(* CODESYS project TeSTL_RECOVERED_2026-06-30T05-16-33.project

Project tree, tasks and I/O mapping:
  Device : CODESYS Control Win V3 x64, CODESYS, version 3.5.22.20
    application Application
      libraries: Standard, 3.5.22.0 (System)
      task MainTask (cyclic, interval t#20ms, priority 1) calls PLC_PRG
      program PLC_PRG [ST]
*)

// Device/Application/PLC_PRG
PROGRAM PLC_PRG
VAR
    // ---- PHYSICAL INPUTS (Mapped to IO Modules) ----
    xProximitySensor     : BOOL;  // Detects a part arriving at the inspection point
    xPartInBin1Sensor    : BOOL;  // Verification sensor for Bin 1
    xPartInBin2Sensor    : BOOL;  // Verification sensor for Bin 2
    xPartInRejectSensor  : BOOL;  // Verification sensor for Reject Bin
    
    // ---- PHYSICAL OUTPUTS (Mapped to Relays/Actuators) ----
    xMainConveyorMotor   : BOOL;  // High-voltage motor running the belt
    xPusherActuator1     : BOOL;  // Pneumatic piston for Bin 1
    xPusherActuator2     : BOOL;  // Pneumatic piston for Bin 2
    
    // ---- RASPBERRY PI NETWORK INTERFACE (Modbus/EtherNET IP Map) ----
    // The Pi writes to these registers
    xPi_Heartbeat        : BOOL;  // Toggle bit to monitor if the Pi is alive
    xPi_NewInstruction   : BOOL;  // Strobe bit signaling a routing decision is ready
    diPi_TargetBin       : DINT;  // Target Destination: 1 = Bin 1, 2 = Bin 2, 3 = Reject
    
    // The PLC writes to these registers for the Pi to read
    xPLC_PartReadyForScan: BOOL;  // Signals the Pi to run its Computer Vision/Camera script
    xPLC_SystemReady     : BOOL;  // System health indicator
    xPLC_ErrorFault      : BOOL;  // Active fault indicator
    
    // ---- INTERNAL CONTROL LOGIC & STATE MACHINE ----
    iSystemState         : INT := 0;   // Main State Machine Step counter
    diAssignedRoute      : DINT;       // Latched routing destination for current part
    tonPusherTimeout     : TON;        // Built-in Timer for Actuator extension
    tonWatchdog          : TON;        // Heartbeat Watchdog Timer for Raspberry Pi communication
    xLastPiHeartbeatState: BOOL;  // Memory flag to track edge transitions of the heartbeat
END_VAR

// ==========================================
// 1. SAFETY & COMMUNICATION WATCHDOG
// ==========================================
// Track if the Raspberry Pi stops communicating. 
// If xPi_Heartbeat doesn't toggle state within 3.0 seconds, trigger a fault.

tonWatchdog(IN := (xPi_Heartbeat = xLastPiHeartbeatState), PT := T#3S);

IF tonWatchdog.Q THEN
    xPLC_ErrorFault := TRUE;
    iSystemState := 99; // Jump straight to Emergency / Fault State
END_IF;

xLastPiHeartbeatState := xPi_Heartbeat; // Store current state for next cyclic scan


// ==========================================
// 2. MAIN SORTING STATE MACHINE
// ==========================================
CASE iSystemState OF
    
    0: (* STATE 0: System Initialization & Idle State *)
        xMainConveyorMotor   := FALSE;
        xPusherActuator1     := FALSE;
        xPusherActuator2     := FALSE;
        xPLC_PartReadyForScan:= FALSE;
        xPLC_SystemReady     := TRUE;
        
        IF NOT xPLC_ErrorFault THEN
            xMainConveyorMotor := TRUE; // Start conveyor if safe
            iSystemState := 10;
        END_IF;

    10: (* STATE 10: Wait for Part Arrival *)
        IF xProximitySensor THEN
            xMainConveyorMotor := FALSE;      // Halt conveyor to take clean camera frame
            xPLC_PartReadyForScan := TRUE;    // Strobe signal to Raspberry Pi
            iSystemState := 20;
        END_IF;

    20: (* STATE 20: Wait for Raspberry Pi Decision Handshake *)
        // Pi processes image -> Writes destination register -> Sets xPi_NewInstruction TRUE
        IF xPi_NewInstruction THEN
            diAssignedRoute := diPi_TargetBin; // Latch the routing decision locally
            xPLC_PartReadyForScan := FALSE;    // Lower the request flag
            xMainConveyorMotor := TRUE;        // Resume conveyor movement
            iSystemState := 30;
        END_IF;

    30: (* STATE 30: Execute Sorting Trajectory *)
        CASE diAssignedRoute OF
            1: (* Route to Bin 1 *)
                xPusherActuator1 := TRUE;
                tonPusherTimeout(IN := TRUE, PT := T#1.5S); // Allow piston to fully extend
                
                IF xPartInBin1Sensor OR tonPusherTimeout.Q THEN
                    xPusherActuator1 := FALSE;
                    tonPusherTimeout(IN := FALSE); // Reset Timer
                    iSystemState := 0;             // Cycle Complete, return to idle
                END_IF;
                
            2: (* Route to Bin 2 *)
                xPusherActuator2 := TRUE;
                tonPusherTimeout(IN := TRUE, PT := T#1.5S);
                
                IF xPartInBin2Sensor OR tonPusherTimeout.Q THEN
                    xPusherActuator2 := FALSE;
                    tonPusherTimeout(IN := FALSE);
                    iSystemState := 0;
                END_IF;
                
            3: (* Route directly to default Reject Bin *)
                IF xPartInRejectSensor THEN
                    iSystemState := 0;
                END_IF;
        ELSE
            // If the Pi passes an invalid destination code, trigger a fault routing anomaly
            xPLC_ErrorFault := TRUE;
            iSystemState := 99;
        END_CASE;

    99: (* STATE 99: Emergency Fault Handling *)
        xMainConveyorMotor   := FALSE;
        xPusherActuator1     := FALSE;
        xPusherActuator2     := FALSE;
        xPLC_SystemReady     := FALSE;
        
        // Auto-recovery mechanism: Clear fault if communication resets and error is acknowledged
        IF NOT tonWatchdog.Q AND NOT xProximitySensor THEN
            xPLC_ErrorFault := FALSE;
            iSystemState := 0;
        END_IF;

END_CASE;

END_PROGRAM
